// Mitsubishi GX Works2 project: 0625(카운트3)   PLC: Q02/Q02H

PROGRAM MAIN
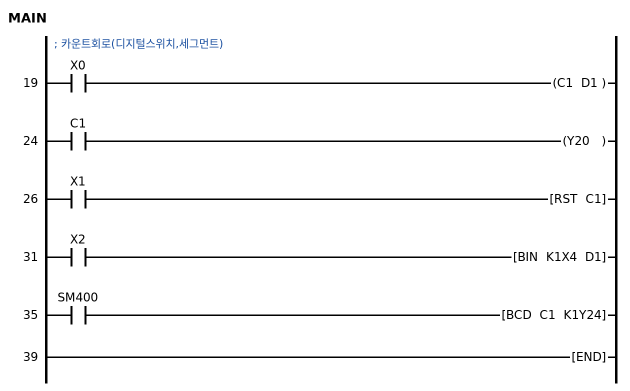
; 카운트회로(디지털스위치,세그먼트)
19    LD      X0
      OUT     C1 D1
24    LD      C1
      OUT     Y20
26    LD      X1
      RST     C1
31    LD      X2
      BIN     K1X4 D1
35    LD      SM400
      BCD     C1 K1Y24
39    END
END_PROGRAM
